{attribute 'GeneratedUsingTerminal: EJ7411-0000-0018'}
{attribute addProperty BoxType "EJ7411-0000-0018"}
{attribute addProperty Id "Target_positionAT %Q*UDINT4"}
{attribute addProperty CRC "86249236"}
{attribute addProperty Size "4"}
TYPE DRV_Target_position_05240F14 :
STRUCT
	{attribute addProperty Name "Target_position"}
	Target_position AT %Q* : UDINT;
END_STRUCT
END_TYPE

(* stored: Version 1.2.0.0, ProductVersion 3.1.4024.9
   DUT DRV_Target_position_05240F14: Id {2c6b2af8-e71b-49cb-ba20-093367080ccc} *)
